FUNCTION_BLOCK FB_ProtectRelay_WIP1 EXTENDS FB_ProtectRelay_Base
VAR_INPUT
						
	
	

END_VAR

VAR_INPUT
	// I/O Inputs 		                                     				
		IN_MesAlarmImax_IO		: BOOL ; // IO max I  fault
		IN_MesAlarmUmin_IO		: BOOL ;  // IO Min U  Fault 
		
END_VAR


VAR
// M_ALARMMNGMT VARIABLES //
                            		
	CmdResetHVCell				: BOOL ; 
	// M_READ VARIABLES//
	
MesDataExd 		    AT %Q*  	: ProtectRelay_WIP1; 	
		


END_VAR

METHOD M_AlarmManagement
VAR 
	// Method local variables (reinitialized at each cycle) 
	FB_AlarmCodeManager : FB_AlarmCodeManager ; 

	ComWarning: BOOL;
	ComAlarm: BOOL;
	KK: BYTE;
	
END_VAR
// Detection Variables

MesDataExd.MesData.MesAlarmImax	:= IN_MesAlarmImax_IO ; 
MesDataExd.MesData.MesAlarmUmin :=  IN_MesAlarmUmin_IO ; 


// ALARM CODE //
	FB_AlarmCodeManager(
		bAlarm1	 := MesDataExd.MesData.MesAlarmImax,// Max I Fault 
		bAlarm2	 := MesDataExd.MesData.MesAlarmUmin,// Min U  Fault
		bAlarm3	 := FALSE, //
		bAlarm4	 := FALSE,//
		bAlarm5	 := FALSE, //
		bAlarm6	 := FALSE,//
		bAlarm7	 := FALSE, //
		bAlarm8	 := FALSE,//
		bAlarm9	 := FALSE, //
		bAlarm10 := FALSE,//
		bAlarm11 := FALSE, //
		bAlarm12 := FALSE,//
		bAlarm13 := FALSE, //
		bAlarm14 := FALSE,//														   
		bAlarm15 := FALSE,//									                      
		wAlarmCode	=>MesDataExd.MesData.MesAlarmCode);


// WARNING CODE //
	FB_AlarmCodeManager(
 		bAlarm1			:= FALSE, //
		bAlarm2			:= FALSE,//
        bAlarm3			:= FALSE, //
		bAlarm4			:= FALSE,// 
		bAlarm5			:= FALSE, // 
		bAlarm6			:= FALSE,// 
		bAlarm7			:= FALSE, // 
		bAlarm8			:= FALSE,// 
		bAlarm9			:= FALSE, // 
		bAlarm10		:= FALSE,// 
		bAlarm11		:= FALSE, // 
		bAlarm12		:= FALSE,//		 
		bAlarm13		:= FALSE,//		 
		bAlarm14		:= FALSE,  //
		bAlarm15		:= FALSE, //
		wAlarmCode	=>MesDataExd.MesData.MesWarningCode);
END_METHOD

METHOD M_Execute

// INITIALIZE // 
	IF bInit THEN
		M_Init() ; 
		bInit		:= FALSE ; 
		
	ELSIF IN_CmdReset_L THEN 
		bInit		:= TRUE ;
		
	END_IF





M_AlarmManagement() ;
END_METHOD

END_FUNCTION_BLOCK

(* stored: Version 1.1.0.1, ProductVersion 3.1.4024.6
   POU FB_ProtectRelay_WIP1: Id {c640a9dc-01b0-4e53-8152-541f5f2dedeb}, SpecialFunc None
   Method M_AlarmManagement: Id {50586635-e794-409b-aa90-06b7a9556803}
   Method M_Execute: Id {ec53dfa2-6fc3-4a59-b8d3-82ea98f1a380} *)
